Staubli VAL3: isActionEmpty.pgx

public program isActionEmpty(bool& x_bEmpty)
begin
  // check if there are some action in the queue
  if aAction.iInstr.sType!="null"
    x_bEmpty=false
  else
    x_bEmpty=true
  endIf
end
